KUKA KRL data list: $config.dat

&ACCESS RV$
&REL 2
DEFDAT $CONFIG
CHAR START_DRAW_FLAG
CHAR START_POINT_FLAG
FRAME ENTRY_POINT_G2
ENDDAT
